SUBAPPLICATION Uebung_011a2 (* Numeric Value Output und BUTTON_PRESS_REPEAT_DONE *)
  (* Standard: 61499-2; Description: Copyright (c) 2023 Meisterschulen am Ostbahnhof This program and the accompanying materials are made available under the terms of the Eclipse Public License 2.0 which is available at https://www.eclipse.org/legal/epl-2.0/ SPDX-License-Identifier: EPL-2.0 *)
  (* Version 1.0, 2023-10-23, Franz Höpfinger, Meisterschulen am Ostbahnhof *)
  IMPORT logiBUS::io::DI::logiBUS_DI;
  IMPORT logiBUS::io::DQ::logiBUS_DO;
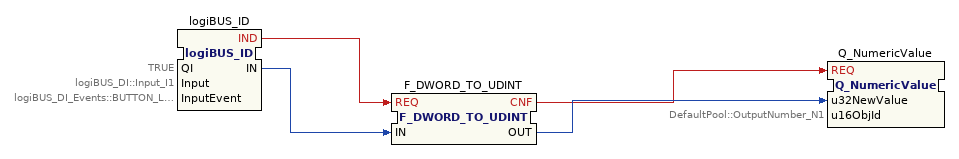
  (* BUTTON_PRESS_UP BUTTON_LONG_PRESS_HOLD BUTTON_LONG_PRESS_UP *)
  FBS
    Q_NumericValue : isobus::ut::Q_NumericValue(u16ObjId := DefaultPool::OutputNumber_N1);
    logiBUS_ID : logiBUS_ID(QI := TRUE, Input := logiBUS_DI::Input_I1, InputEvent := logiBUS_DI_Events::BUTTON_LONG_PRESS_UP);
    F_DWORD_TO_UDINT : F_DWORD_TO_UDINT;
  END_FBS
  EVENT_CONNECTIONS
    logiBUS_ID.IND TO F_DWORD_TO_UDINT.REQ;
    F_DWORD_TO_UDINT.CNF TO Q_NumericValue.REQ;
  END_CONNECTIONS
  DATA_CONNECTIONS
    logiBUS_ID.IN TO F_DWORD_TO_UDINT.IN;
    F_DWORD_TO_UDINT.OUT TO Q_NumericValue.u32NewValue;
  END_CONNECTIONS
END_SUBAPPLICATION
